// TIA Portal V19 export
TYPE "LAF_typeAxisDiagStatusWord"
TITLE = LAF_typeAxisDiagStatusWord
// Status information of a Technology object
// stored: Access Published
   STRUCT
      bit00_Enable { ExternalWritable := 'False'} : Bool;   // Enable status. The technology object has been enabled / Enable
      bit01_Error { ExternalWritable := 'False'} : Bool;   // An error is present / Error
      bit02_RestartActive { ExternalWritable := 'False'} : Bool;   // A restart is active. The technology object will be reinitialized / RestartActive
      bit03_OnlineStartValuesChanged { ExternalWritable := 'False'} : Bool;   // The restart tags have been changed. For the changes to be applied, the thechnogy object must be reinitialized / OnlineStartValuesChanged
      bit04_ControlPanelActive { ExternalWritable := 'False'} : Bool;   // The axis control panel is active / ControlPanelActive
      bit05_HomingDone { ExternalWritable := 'False'} : Bool;   // Homing status. The technology object is homed / HomingDone
      bit06_Done { ExternalWritable := 'False'} : Bool;   // Done. No motion job is in progress and the axis control panel is deactivated / Done
      bit07_Standstill { ExternalWritable := 'False'} : Bool;   // Standstill signal. The axis is at a standstill / StandStill
      bit08_PositioningCommand { ExternalWritable := 'False'} : Bool;   // A positioning command is active ("MC_MoveRelative","MC_MoveAbsolute") / PositioningCommand
      bit09_JogCommand { ExternalWritable := 'False'} : Bool;   // An "MC_MoveJog" job is running / JogCommand
      bit10_VelocityCommand { ExternalWritable := 'False'} : Bool;   // An "MC_MoveVelocity" job is running / VelocityCommand
      bit11_HomingCommand { ExternalWritable := 'False'} : Bool;   // An "MC_Home" job is being processed / HomingCommand
      bit12_ConstantVelocity { ExternalWritable := 'False'} : Bool;   // The velocity setpoint is reached. A constant velocity setpoint is output / ConstantVelocity
      bit13_Accelerating { ExternalWritable := 'False'} : Bool;   // An acceleration operation is active / Accelerating
      bit14_Decelerating { ExternalWritable := 'False'} : Bool;   // A deacceleration operation is active / Decelerating
      bit15_SWLimitMinActive { ExternalWritable := 'False'} : Bool;   // A negative software limit switch has been approached or exceeded / SWLimitMinActive
      bit16_SWLimitMaxActive { ExternalWritable := 'False'} : Bool;   // A positive software limit switch has been approached or exceeded / SWLimitMaxActive
      bit17_HWLimitMinActive { ExternalWritable := 'False'} : Bool;   // A negative hardware limit switch has been approached or exceeded / HWLimitMinActive
      bit18_HWLimitMaxActive { ExternalWritable := 'False'} : Bool;   // A positive hardware limit switch has been approached or exceeded / HWLimitMaxActive
      bit19_Reserved { ExternalWritable := 'False'} : Bool;   // Reserved
      bit20_Reserved { ExternalWritable := 'False'} : Bool;   // Reserved
      bit21_Synchronizing { ExternalWritable := 'False'} : Bool;   // The axis synchronizes to a leading value / Synchronizing
      bit22_Synchronous { ExternalWritable := 'False'} : Bool;   // The axis moves synchronously to a leading value / Synhronous
      bit23_SuperimposedMotionCommand { ExternalWritable := 'False'} : Bool;   // An "MC_MoveSuperimposed" job is running / SuperimposedMotionCommand
      bit24_PhasingCommand { ExternalWritable := 'False'} : Bool;   // An "MC_PhasingAbsolute" or "MC_PhasingRelative" job for the leading value offset is active / PhasingCommand
      bit25_AxisSimulation { ExternalWritable := 'False'} : Bool;   // The technology object is in simulation / AxisSimulation
      bit26_TorqueLimitingCommand { ExternalWritable := 'False'} : Bool;   // An "MC_TorqueLimiting" job is running / TorqueLimitingCommand
      bit27_InLimitation { ExternalWritable := 'False'} : Bool;   // The drive operates at least at the threshold value (default 90%) of the torque limit/force limitation / InLimitation
      bit28_NonPositionControlled { ExternalWritable := 'False'} : Bool;   // The axis is not in position-controlled mode / NonPositionControlled
      bit29_KinematicsMotionCommand { ExternalWritable := 'False'} : Bool;   // The axis is used for a kinematics job / Reserved
      bit30_InClamping { ExternalWritable := 'False'} : Bool;   // The axis is clamped at a fixed stop / InClamping
      bit31_MotionInCommand { ExternalWritable := 'False'} : Bool;   // A "MC_MotionIn" job is running / Reserved
   END_STRUCT;
END_TYPE
